FUNCTION_BLOCK FB_Fanuc
VAR_INPUT
END_VAR
VAR_OUTPUT
END_VAR
VAR
END_VAR

END_FUNCTION_BLOCK

(* stored: Version 1.1.0.1, ProductVersion 3.1.4024.9
   POU FB_Fanuc: Id {12ac1ec7-c492-4001-99fb-5b6278171b1a}, SpecialFunc None *)
